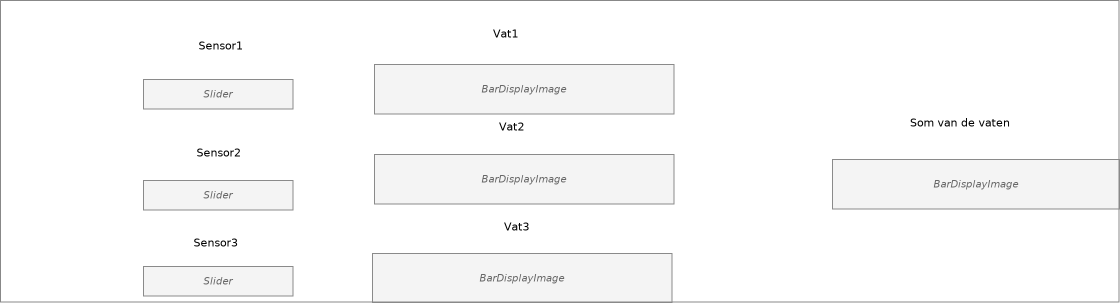
VISUALIZATION Visualization  // 1120x303
    Slider (143,79 150x30), variable: MAIN.nSensor1, scale 0..2000
    Slider (143,180 150x30), variable: MAIN.nSensor2, scale 0..3000
    Slider (143,266 150x30), variable: MAIN.nSensor3, scale 0..5000
    BarDisplayImage (374,64 300x50), value: MAIN.nVat1, style: BarDisplayImage-Gray, scale format: %.1f, scale 0..100
    BarDisplayImage (832,159 288x50), value: MAIN.nBardisplay, style: BarDisplayImage-Gray, scale format: %.1f, scale 0..300
    BarDisplayImage (374,154 300x50), value: MAIN.nVat2, style: BarDisplayImage-Gray, scale format: %.1f, scale 0..100
    BarDisplayImage (372,253 300x50), value: MAIN.nVat3, style: BarDisplayImage-Gray, scale format: %.1f, scale 0..100
    Label (146,31 150x30), "Sensor1"
    Label (144,138 150x30), "Sensor2"
    Label (141,228 150x30), "Sensor3"
    Label (431,19 150x30), "Vat1"
    Label (437,112 150x30), "Vat2"
    Label (442,212 150x30), "Vat3"
    Label (885,108 150x30), "Som van de vaten"
END_VISUALIZATION

(* stored: Version 1.1.0.1, ProductVersion 3.1.4024.12
   Visu Visualization: Id {a8fb7c22-8322-482d-8b07-477d731ce135} *)
